Staubli VAL3: FCheckInBox1Pos.pgx

public program FCheckInBox1Pos(tool t_tool, frame fr_frame, bool& b_inArea[], num& x_nKeyNum[], num& nTolKeyNum[])
// Pruefen ob Roboter innerhalb eines definierten Bereichs
  local trsf tr_here
  local point p_here
  local trsf tr_NegPos
  local trsf tr_PosPos
  local trsf tr_BoxPos1
  local trsf tr_BoxPos2
begin
  //Header
  if false
    //判断机器人是否属于所设定的空间盒子中
    //Parameter:
    //  p_BoxPos1: Position 1 (包括开始位置跟结束位置)
    //  p_BoxPos2: Position 2 (包括开始位置跟结束位置)
    //  b_inArea: 返回参数  true  : 机器人在矩形中
    //                          false : 机器人属于非矩形中
    //
  endIf
  //判断变量返回
  b_inArea=true
  p_here=here(t_tool,fr_frame)
  tr_here=p_here.trsf
  if (tr_here.x>(x_nKeyNum[3]+nTolKeyNum[3])) or (tr_here.y>(x_nKeyNum[4]+nTolKeyNum[4])) or (tr_here.z>(x_nKeyNum[5]+nTolKeyNum[5]))
    b_inArea=false
  endIf
  if (tr_here.x<(x_nKeyNum[0]-nTolKeyNum[0])) or (tr_here.y<(x_nKeyNum[1]-nTolKeyNum[1])) or (tr_here.z<(x_nKeyNum[2]-nTolKeyNum[2]))
    b_inArea=false
  endIf
end
